FUNCTION FsF_IecApplicationInformation : ITcIecApplicationInfo

FW_ObjMgr_GetObjectInstance(TwinCAT_SystemInfoVarList._AppInfo.ObjId, TC_GLOBAL_IID_LIST.IID_ITcIecApplicationInfo, ADR(FsF_IecApplicationInformation));

END_FUNCTION

(* stored: Version 1.1.0.1, ProductVersion 3.1.4024.4
   POU FsF_IecApplicationInformation: Id {c801c14f-c7fb-4dfb-a113-f15126d5b18d}, SpecialFunc None *)
